Staubli VAL3: showBoolStatus.pgx

public program showBoolStatus(bool x_bStatus (dimensions=1), string& x_sEvent[] (dimensions=1))
begin
  if x_bStatus
    x_sEvent="[x]"
  else
    x_sEvent="[ ]"
  endIf
end
